Yaskawa INFORM job: UROS.JBI

/JOB
//NAME UROS
//POS
///NPOS 0,0,0,1,0,0
///TOOL 1
///POSTYPE BASE
///RECTAN
///RCONF 1,0,0,0,0,0,0,0,0,0,0,0,0,0,0,0,0,0,0,0,0,0,0,0
P00000=165.804,1062.206,913.968,179.6354,10.9678,-179.8406
//INST
///DATE 2019/10/04 13:40
///ATTR SC,RW
///GROUP1 RB1
NOP
GETS PX000 $PX000
CNVRT PX000 PX000 UF#(1)
SUB P000 P000
CNVRT PX000 PX000 BF
END
